// TIA Portal project "Game" (V18)

(* hardware
DEVICE "S7-1200 station_1"  S7-1200 Station
   slot 0: "Rack_0"  S7-1200 Rack  Rack  V1.0
   slot 1: "PLC_1"  CPU 1215C DC/DC/DC  6ES7 215-1AG40-0XB0  V4.4
DEVICE "PC-System_1"  SIMATIC PC station
   slot 0: "SIMATIC PC station"  Rail  SIMATIC PC-Station  V1.0
      slot 125: "Stationmanager"  Station_Manager  V6.0.4
   slot 1: "IE general_1"  IE General  IE_CP  V8.2.0
   slot 2: "HMI_RT_1"  WinCC RT Advanced  6AV2 104-0xxxx-xxxx  16.0.0.0
      slot 33792: "Computer interface"  Host interface
*)

// ===== PLC "PLC_1"  CPU 1215C DC/DC/DC =====

VAR_GLOBAL   // PLC tag table "Default tag table"
   "System_Byte" AT %MB1 : Byte;   // System Byte used for diagnostics or system status.
   "FirstScan" AT %M1.0 : Bool;   // Indicates the first scan of the PLC program.
   "DiagStatusUpdate" AT %M1.1 : Bool;   // Trigger for updating diagnostic status.
   "AlwaysTRUE" AT %M1.2 : Bool;   // Always holds the value TRUE.
   "AlwaysFALSE" AT %M1.3 : Bool;   // Always holds the value FALSE.
   "Clock_Byte" AT %MB0 : Byte;   // System clock byte for generating clock pulses.
   "Clock_10Hz" AT %M0.0 : Bool;   // 10 Hz clock pulse for timing operations.
   "Clock_5Hz" AT %M0.1 : Bool;   // 5 Hz clock pulse for timing operations.
   "Clock_2.5Hz" AT %M0.2 : Bool;   // 2.5 Hz clock pulse for timing operations.
   "Clock_2Hz" AT %M0.3 : Bool;   // 2 Hz clock pulse for timing operations.
   "Clock_1.25Hz" AT %M0.4 : Bool;   // 1.25 Hz clock pulse for timing operations.
   "Clock_1Hz" AT %M0.5 : Bool;   // 1 Hz clock pulse for timing operations.
   "Clock_0.625Hz" AT %M0.6 : Bool;   // 0.625 Hz clock pulse for timing operations.
   "Clock_0.5Hz" AT %M0.7 : Bool;   // 0.5 Hz clock pulse for timing operations.
   "lifebit" AT %M5.0 : Bool;   // Life bit toggled for system health monitoring.
   "Tag_1" AT %MW11 : Int;   // Temporary tag for integer calculations.
   "Tag_2" AT %MW12 : Word;   // Temporary tag for word calculations.
   "Tag_3" AT %M14.0 : Bool;   // Auxiliary flag for custom logic.
   "Tag_4" AT %MW4 : Word;   // Temporary tag for word operations.
   "draw number" AT %M20.0 : Bool;   // Trigger for generating random numbers.
   "Tag_6" AT %M100.0 : Bool;   // Auxiliary flag for random number validation.
   "temp int" AT %MW1 : Int;   // Temporary integer for calculations.
   "new game" AT %M15.0 : Bool;   // Signal to initialize a new game.
   "Tag_5" AT %M100.1 : Bool;   // Auxiliary flag for game initialization.
   "Tag_7" AT %M61.0 : Bool;   // Auxiliary signal for internal processing.
   "Tag_8" AT %M16.0 : Bool;   // Auxiliary signal for click detection.
   "Tag_9" AT %M16.1 : Bool;   // Auxiliary signal for click detection.
   "Tag_10" AT %M120.1 : Bool;   // Auxiliary signal for internal processing.
   "Tag_11" AT %M45.0 : Bool;   // Flag for triggering game logic.
   "Tag_12" AT %M45.1 : Bool;   // Auxiliary signal for additional logic.
   "reset limit" AT %M50.0 : Bool;   // Resets the field discovery limit.
   "start timer" AT %M40.0 : Bool;   // Starts the timer for incorrect moves.
   "start timer 2" AT %M40.1 : Bool;   // Starts the timer for correct moves.
   "running" AT %M10.5 : Bool;   // Indicates that the game is currently running.
   "win" AT %M10.6 : Bool;   // Signals that the game has been won.
   "Click1" AT %M65.0 : Bool;   // Signal for the first tile click.
   "Click2" AT %M65.1 : Bool;   // Signal for the second tile click.
   "Click3" AT %M65.2 : Bool;   // Signal for the third tile click.
   "Click4" AT %M65.3 : Bool;   // Signal for the fourth tile click.
   "Click5" AT %M65.4 : Bool;   // Signal for the fifth tile click.
   "Click6" AT %M65.5 : Bool;   // Signal for the sixth tile click.
   "Click7" AT %M65.6 : Bool;   // Signal for the seventh tile click.
   "Click8" AT %M65.7 : Bool;   // Signal for the eighth tile click.
   "Click9" AT %M66.0 : Bool;   // Signal for the ninth tile click.
   "Click10" AT %M66.1 : Bool;   // Signal for the tenth tile click.
   "Click11" AT %M66.2 : Bool;   // Signal for the eleventh tile click.
   "Click12" AT %M66.3 : Bool;   // Signal for the twelfth tile click.
   "Click13" AT %M66.4 : Bool;   // Signal for the thirteenth tile click.
   "Click14" AT %M66.5 : Bool;   // Signal for the fourteenth tile click.
   "Click15" AT %M66.6 : Bool;   // Signal for the fifteenth tile click.
   "Click16" AT %M66.7 : Bool;   // Signal for the sixteenth tile click.
END_VAR

DATA_BLOCK "Data_block_1"   // DB1
{ S7_Optimized_Access := 'TRUE' }
VERSION : 0.1
   VAR
      "time" : DTL;   // Current date and time used for generating random numbers.
      time2 : Time_Of_Day;   // Converted time of day extracted from the current system time.
      "time on udint" : UDInt;   // System time in unsigned double integer format for easier calculations.
      "tile array hidden" : Array[1..16] of Int;   // Stores the hidden values for each tile in the game.
      "tile array" : Array[1..16] of Int;   // Stores the currently revealed values for each tile.
      "guess tiles" : Array[1..16] of Int;   // Used to track player's guesses during the game
      "random number" : Int;   // Holds the latest randomly generated number for assigning tiles.
      "random numbers" : Array[1..16] of Int;   // Array of all unique randomly generated numbers for the game tiles.
      "array filled" : Bool;   // Indicates whether the tile array hidden is fully initialized.
      "number of moves" : Int;   // Tracks the total number of moves made by the player.
      "click detection" : Array[1..16] of Bool;   // Detects if a tile has been clicked by the player.
      "click detection2" : Array[1..16] of Bool;   // Additional array for detecting tile clicks used during validation.
      "field discovery limit" : Int;   // Counts the number of fields discovered by the player during a turn.
      "end of incorrect move" : Bool;   // Signals the end of an incorrect move.
      "end of correct move" : Bool;   // Signals the end of a correct move.
      "comparison mode" : Bool;   // Enables or disables the comparison logic between selected tiles.
      value1 : Int;   // The value of the first selected tile during a player's turn.
      value2 : Int;   // The value of the second selected tile during a player's turn.
      "value1 idx" : Int;   // The index of the first selected tile in the tile array.
      "value2 idx" : Int;   // The index of the second selected tile in the tile array.
      flag1 : Bool;   // Trigger used for checking game logic events like tile selection.
      flag2 : Bool;   // Additional trigger for handling specific game logic.
   END_VAR
BEGIN
END_DATA_BLOCK

// folder: System blocks/Program resources

DATA_BLOCK "IEC_Counter_0_DB"   // DB2
{ S7_Optimized_Access := 'TRUE' }
AUTHOR : Simatic
FAMILY : IEC
NAME : CNTR
VERSION : 1.0
// stored: InstanceOfName IEC_COUNTER
"IEC_COUNTER"
BEGIN
END_DATA_BLOCK

DATA_BLOCK "IEC_Timer_0_DB_2"   // DB4
{ S7_Optimized_Access := 'TRUE' }
AUTHOR : Simatic
FAMILY : IEC
NAME : IEC_TMR
VERSION : 1.0
// stored: InstanceOfName IEC_TIMER
"IEC_TIMER"
BEGIN
END_DATA_BLOCK

DATA_BLOCK "IEC_Timer_0_DB"   // DB5
{ S7_Optimized_Access := 'TRUE' }
AUTHOR : Simatic
FAMILY : IEC
NAME : IEC_TMR
VERSION : 1.0
// stored: InstanceOfName IEC_TIMER
"IEC_TIMER"
BEGIN
END_DATA_BLOCK

// folder: (top level)

FUNCTION "board filling SCL" : Void   // FC6, SCL
TITLE = board filling SCL
{ S7_Optimized_Access := 'TRUE' }
AUTHOR : krist
VERSION : 0.1
// Generating and placing random numbers on the game board.
   VAR_TEMP
      new : Bool;
      temp1 : Int;
      temp2 : Int;
      temp3 : Int;
      temp4 : Int;
   END_VAR
BEGIN
   #temp2 := 1;  // Iniciē mainīgo, kas skaita aizpildītās vērtības "random numbers" masīvā

   // Galvenais cikls, kas atkārto procesu 8 reizes
   FOR #temp1 := 1 TO 8 DO

       // Pārbauda, vai izlozētais skaitlis jau ir izmantots
       #"new" := FALSE;
       WHILE #"new" <> TRUE DO

           // Izveido nejaušu skaitli, izmantojot sistēmas laiku
           "Tag_1" := RD_LOC_T("Data_block_1"."time");
           "Data_block_1".time2 := DTL_TO_TOD("Data_block_1"."time");
           "Data_block_1"."time on udint" := TOD_TO_UDINT("Data_block_1".time2);
           "Data_block_1"."random number" := "Data_block_1"."time on udint" MOD 16;  // Ģenerē nejaušu skaitli starp 0 un 15
           "Data_block_1"."random number" += 1;  // Pielāgo, lai intervāls būtu no 1 līdz 16

           #"new" := TRUE;  // Pieņem, ka skaitlis ir jauns

           // Pārbauda, vai skaitlis jau eksistē "random numbers" masīvā
           FOR #temp3 := 1 TO 16 DO
               IF "Data_block_1"."random number" = "Data_block_1"."random numbers"[#temp3] THEN
                   #"new" := FALSE;  // Ja skaitlis eksistē, atkārto ģenerēšanas procesu
                   EXIT;
               END_IF;
           END_FOR;

       END_WHILE;

       // Piešķir nejaušo vērtību "tile array hidden" un saglabā "random numbers" masīvā
       "Data_block_1"."tile array hidden"["Data_block_1"."random number"] := #temp1;
       "Data_block_1"."random numbers"[#temp2] := "Data_block_1"."random number";
       #temp2 += 1;  // Palielina aizpildīto vērtību skaitītāju

       // Pārbauda, vai visi 16 skaitļi ir aizpildīti
       IF #temp2 = 16 THEN
           FOR #temp4 := 1 TO 16 DO
               IF "Data_block_1"."tile array hidden"[#temp4] = 0 THEN
                   "Data_block_1"."tile array hidden"[#temp4] := #temp1;  // Aizpilda atlikušo vietu masīvā
                   EXIT;
               END_IF;
           END_FOR;
           EXIT;  // Iziet no galvenā cikla, ja visi skaitļi ir aizpildīti
       END_IF;

       // Pārbauda, vai izlozētais skaitlis jau ir izmantots (otra izloze)
       #"new" := FALSE;
       WHILE #"new" <> TRUE DO

           // Izveido nejaušu skaitli, izmantojot sistēmas laiku
           "Tag_1" := RD_LOC_T("Data_block_1"."time");
           "Data_block_1".time2 := DTL_TO_TOD("Data_block_1"."time");
           "Data_block_1"."time on udint" := TOD_TO_UDINT("Data_block_1".time2);
           "Data_block_1"."random number" := "Data_block_1"."time on udint" MOD 15;  // Ģenerē nejaušu skaitli starp 0 un 14
           "Data_block_1"."random number" += 1;  // Pielāgo, lai intervāls būtu no 1 līdz 15

           #"new" := TRUE;  // Pieņem, ka skaitlis ir jauns

           // Pārbauda, vai skaitlis jau eksistē "random numbers" masīvā
           FOR #temp3 := 1 TO 16 DO
               IF "Data_block_1"."random number" = "Data_block_1"."random numbers"[#temp3] THEN
                   #"new" := FALSE;  // Ja skaitlis eksistē, atkārto ģenerēšanas procesu
                   EXIT;
               END_IF;
           END_FOR;

       END_WHILE;

       // Piešķir nejaušo vērtību "tile array hidden" un saglabā "random numbers" masīvā
       "Data_block_1"."tile array hidden"["Data_block_1"."random number"] := #temp1;
       "Data_block_1"."random numbers"[#temp2] := "Data_block_1"."random number";
       #temp2 += 1;  // Palielina aizpildīto vērtību skaitītāju

   END_FOR;

   // Atzīmē, ka masīvs ir pilnībā aizpildīts
   "Data_block_1"."array filled" := true;
END_FUNCTION

FUNCTION "clearing memory SCL" : Void   // FC7, SCL
TITLE = clearing memory SCL
{ S7_Optimized_Access := 'TRUE' }
AUTHOR : krist
VERSION : 0.1
// Clearing the game arrays and restoring the initial state
   VAR_TEMP
      temp : Int;
   END_VAR
BEGIN
   // Inicializē masīvus un mainīgos
   FOR #temp := 1 TO 16 DO
       "Data_block_1"."tile array"[#temp] := 0;           // Notīra "tile array" masīvu, uzstādot vērtības uz 0
       "Data_block_1"."tile array hidden"[#temp] := 0;    // Notīra "tile array hidden" masīvu, uzstādot vērtības uz 0
       "Data_block_1"."random numbers"[#temp] := 0;       // Notīra "random numbers" masīvu, uzstādot vērtības uz 0
       "Data_block_1"."click detection"[#temp] := 0;      // Notīra "click detection" masīvu, uzstādot vērtības uz 0
   END_FOR;

   // Inicializē citus parametrus
   "Data_block_1"."array filled" := FALSE;   // Norāda, ka masīvs nav aizpildīts
   "Data_block_1"."number of moves" := 0;    // Uzstāda gājienu skaitu uz 0
   "Data_block_1".value1 := 0;               // Notīra vērtību 1
   "Data_block_1".value2 := 0;               // Notīra vērtību 2
   "Data_block_1"."value1 idx" := 0;         // Notīra pirmā elementa indeksu
   "Data_block_1"."value2 idx" := 0;         // Notīra otrā elementa indeksu

   "Data_block_1"."comparison mode" := FALSE; // Izslēdz salīdzināšanas režīmu
   "win" := FALSE;                            // Norāda, ka spēle vēl nav uzvarēta
END_FUNCTION

FUNCTION "game SCL" : Void   // FC8, SCL
TITLE = game SCL
{ S7_Optimized_Access := 'TRUE' }
AUTHOR : krist
VERSION : 0.1
// The core logic of the game, including click processing and comparison.
   VAR_TEMP
      first : Int;
      second : Int;
   END_VAR
BEGIN

   "reset limit" := FALSE;  // Atjaunot limitu tiek atslēgts

   // Pārbaude, vai "field discovery limit" ir mazāks vai vienāds ar 2 un "Tag_11" ir TRUE
   IF "Data_block_1"."field discovery limit" <= 2 AND "Tag_11" THEN
       // Pārbauda katru elementu "click detection2" masīvā
       FOR #first := 1 TO 16 DO
           IF "Data_block_1"."click detection2"[#first] = TRUE AND "Data_block_1".value1 = 0 THEN
               EXIT;  // Iziet no cikla, ja atklāts klikšķis un vērtība 1 ir 0
           END_IF;
       END_FOR;

       // Apstrādā klikšķus un saglabā vērtības
       FOR #first := 1 TO 16 DO
           IF "Data_block_1"."click detection2"[#first] = TRUE THEN
               "Data_block_1"."tile array"[#first] := "Data_block_1"."tile array hidden"[#first];  // Atklāj slēpto elementu

               IF "Data_block_1".value1 = 0 THEN
                   "Data_block_1".value1 := "Data_block_1"."tile array"[#first];  // Saglabā pirmo vērtību
                   "Data_block_1"."value1 idx" := #first;  // Saglabā pirmā elementa indeksu
               END_IF;

               "Data_block_1".value2 := "Data_block_1"."tile array"[#first];  // Saglabā otro vērtību
               "Data_block_1"."value2 idx" := #first;  // Saglabā otrā elementa indeksu
           END_IF;
       END_FOR;
   END_IF;

   // Aktivizē trigeri, ja "field discovery limit" ir vienāds ar 2
   "R_TRIG_DB"(CLK := "Data_block_1"."field discovery limit" = 2,
               Q => "Data_block_1".flag1);

   // Ja trigeris aktivizēts, palielina gājienu skaitu
   IF "Data_block_1".flag1 = TRUE THEN
       "Data_block_1"."number of moves" += 1;

       // Pārbauda, vai vērtības ir vienādas
       IF "Data_block_1".value1 = "Data_block_1".value2 THEN
           "start timer 2" := TRUE;  // Aktivizē otro taimeri
       ELSE
           "start timer" := TRUE;  // Aktivizē pirmo taimeri
       END_IF;
   END_IF;

   // Apstrādā nepareizo gājienu
   IF "Data_block_1"."end of incorrect move" THEN
       "start timer" := FALSE;  // Izslēdz taimeri

       // Atiestata klikšķu izvēlētās vērtības un pozīcijas
       "Data_block_1"."tile array"["Data_block_1"."value1 idx"] := 0;
       "Data_block_1"."tile array"["Data_block_1"."value2 idx"] := 0;
       "Data_block_1".value1 := 0;
       "Data_block_1".value2 := 0;
       "Data_block_1"."value1 idx" := 0;
       "Data_block_1"."value2 idx" := 0;

       "reset limit" := TRUE;  // Aktivizē limitu
   END_IF;

   // Apstrādā pareizo gājienu
   IF "Data_block_1"."end of correct move" THEN
       "start timer 2" := FALSE;  // Izslēdz otro taimeri

       // Atiestata klikšķu izvēlētās vērtības un pozīcijas
       "Data_block_1".value1 := 0;
       "Data_block_1".value2 := 0;
       "Data_block_1"."value1 idx" := 0;
       "Data_block_1"."value2 idx" := 0;

       "reset limit" := TRUE;  // Aktivizē limitu
   END_IF;

   // Pārbauda, vai visi elementi ir atklāti
   FOR #second := 1 TO 16 DO
       IF "Data_block_1"."tile array"[#second] = 0 THEN
           EXIT;  // Iziet, ja kāds elements nav atklāts
       END_IF;

       IF #second = 16 THEN
           "win" := TRUE;  // Uzvaras nosacījums
       END_IF;
   END_FOR;

   // Atiestata klikšķu detekcijas statusu
   FOR #first := 1 TO 16 DO
       "Data_block_1"."click detection2"[#first] := FALSE;
   END_FOR;
END_FUNCTION

FUNCTION "button operation LAD" : Void   // FC9, LAD
TITLE = button operation LAD
{ S7_Optimized_Access := 'TRUE' }
AUTHOR : krist
VERSION : 0.1
// Detecting clicks and passing them to game logic.
   VAR_TEMP   // added for the SCL form of the ladder/FBD networks
      _w1 : Bool;
      _w2 : Bool;
      _w3 : Bool;
      _w4 : Bool;
      _w5 : Bool;
      _w6 : Bool;
      _w7 : Bool;
      _w8 : Bool;
      _w9 : Bool;
      _w10 : Bool;
      _w11 : Bool;
      _w12 : Bool;
      _w13 : Bool;
      _w14 : Bool;
      _w15 : Bool;
      _w16 : Bool;
      _w17 : Bool;
      _w18 : Bool;
   END_VAR
BEGIN

REGION Network 1: Additional array for detecting tile clicks used during validation.
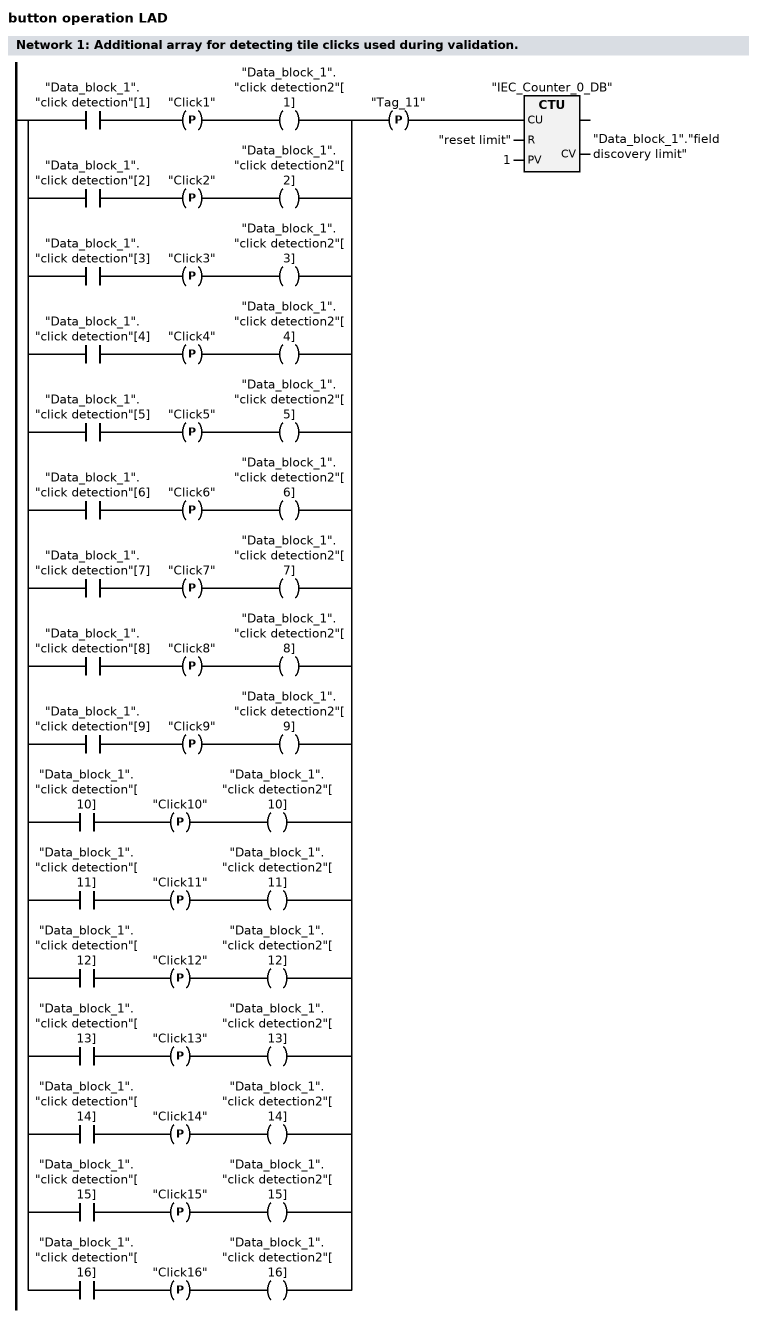
   #_w1 := "Data_block_1"."click detection"[1] AND NOT "Click1";   // rising edge
   "Click1" := "Data_block_1"."click detection"[1];
   "Data_block_1"."click detection2"[1] := #_w1;
   #_w2 := "Data_block_1"."click detection"[2] AND NOT "Click2";   // rising edge
   "Click2" := "Data_block_1"."click detection"[2];
   "Data_block_1"."click detection2"[2] := #_w2;
   #_w3 := "Data_block_1"."click detection"[3] AND NOT "Click3";   // rising edge
   "Click3" := "Data_block_1"."click detection"[3];
   "Data_block_1"."click detection2"[3] := #_w3;
   #_w4 := "Data_block_1"."click detection"[4] AND NOT "Click4";   // rising edge
   "Click4" := "Data_block_1"."click detection"[4];
   "Data_block_1"."click detection2"[4] := #_w4;
   #_w5 := "Data_block_1"."click detection"[5] AND NOT "Click5";   // rising edge
   "Click5" := "Data_block_1"."click detection"[5];
   "Data_block_1"."click detection2"[5] := #_w5;
   #_w6 := "Data_block_1"."click detection"[6] AND NOT "Click6";   // rising edge
   "Click6" := "Data_block_1"."click detection"[6];
   "Data_block_1"."click detection2"[6] := #_w6;
   #_w7 := "Data_block_1"."click detection"[7] AND NOT "Click7";   // rising edge
   "Click7" := "Data_block_1"."click detection"[7];
   "Data_block_1"."click detection2"[7] := #_w7;
   #_w8 := "Data_block_1"."click detection"[8] AND NOT "Click8";   // rising edge
   "Click8" := "Data_block_1"."click detection"[8];
   "Data_block_1"."click detection2"[8] := #_w8;
   #_w9 := "Data_block_1"."click detection"[9] AND NOT "Click9";   // rising edge
   "Click9" := "Data_block_1"."click detection"[9];
   "Data_block_1"."click detection2"[9] := #_w9;
   #_w10 := "Data_block_1"."click detection"[10] AND NOT "Click10";   // rising edge
   "Click10" := "Data_block_1"."click detection"[10];
   "Data_block_1"."click detection2"[10] := #_w10;
   #_w11 := "Data_block_1"."click detection"[11] AND NOT "Click11";   // rising edge
   "Click11" := "Data_block_1"."click detection"[11];
   "Data_block_1"."click detection2"[11] := #_w11;
   #_w12 := "Data_block_1"."click detection"[12] AND NOT "Click12";   // rising edge
   "Click12" := "Data_block_1"."click detection"[12];
   "Data_block_1"."click detection2"[12] := #_w12;
   #_w13 := "Data_block_1"."click detection"[13] AND NOT "Click13";   // rising edge
   "Click13" := "Data_block_1"."click detection"[13];
   "Data_block_1"."click detection2"[13] := #_w13;
   #_w14 := "Data_block_1"."click detection"[14] AND NOT "Click14";   // rising edge
   "Click14" := "Data_block_1"."click detection"[14];
   "Data_block_1"."click detection2"[14] := #_w14;
   #_w15 := "Data_block_1"."click detection"[15] AND NOT "Click15";   // rising edge
   "Click15" := "Data_block_1"."click detection"[15];
   "Data_block_1"."click detection2"[15] := #_w15;
   #_w16 := "Data_block_1"."click detection"[16] AND NOT "Click16";   // rising edge
   "Click16" := "Data_block_1"."click detection"[16];
   "Data_block_1"."click detection2"[16] := #_w16;
   #_w17 := #_w1 OR #_w2 OR #_w3 OR #_w4 OR #_w5 OR #_w6 OR #_w7 OR #_w8 OR #_w9 OR #_w10 OR #_w11 OR #_w12 OR #_w13 OR #_w14 OR #_w15 OR #_w16;
   #_w18 := #_w17 AND NOT "Tag_11";   // rising edge
   "Tag_11" := #_w17;
   "IEC_Counter_0_DB".CTU(CU := #_w18,
                          R := "reset limit",
                          PV := 1,
                          CV => "Data_block_1"."field discovery limit");
END_REGION
END_FUNCTION

FUNCTION "timer LAD" : Void   // FC10, LAD
TITLE = timer LAD
{ S7_Optimized_Access := 'TRUE' }
VERSION : 0.1
// Timer functions for handling correct and incorrect moves.
BEGIN

REGION Network 1: Signals the end of an incorrect move.
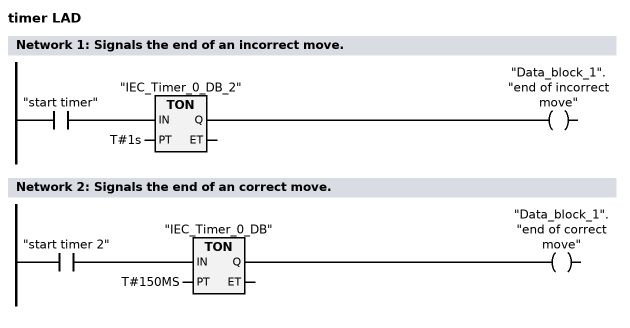
   "IEC_Timer_0_DB_2".TON(IN := "start timer", PT := T#1s);
   "Data_block_1"."end of incorrect move" := "IEC_Timer_0_DB_2".Q;
END_REGION

REGION Network 2: Signals the end of an correct move.
   "IEC_Timer_0_DB".TON(IN := "start timer 2", PT := T#150MS);
   "Data_block_1"."end of correct move" := "IEC_Timer_0_DB".Q;
END_REGION
END_FUNCTION

ORGANIZATION_BLOCK "Main"   // OB1, LAD, ProgramCycle
TITLE = "Main Program Sweep (Cycle)"
{ S7_Optimized_Access := 'TRUE' }
VERSION : 0.1
   VAR_INPUT
      Initial_Call : Bool;   // Initial call of this OB
      Remanence : Bool;   // =True, if remanent data are available
   END_VAR
   VAR_TEMP   // added for the SCL form of the ladder/FBD networks
      _w1 : Bool;
      _w2 : Bool;
   END_VAR
BEGIN

REGION Network 1
   // indicates systems activity
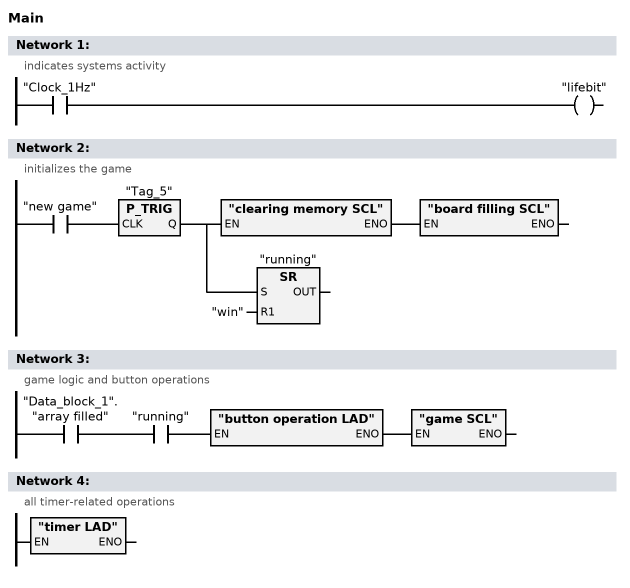
   RUNG wire#powerrail
      Contact( "Clock_1Hz" )
      Coil( "lifebit" )
   END_RUNG
   // the same network as SCL:
   "lifebit" := "Clock_1Hz";
END_REGION

REGION Network 2
   // initializes the game
   RUNG wire#powerrail
      Contact( "new game" )
      P_Trig( "Tag_5" )
      wire#w1
      "clearing memory SCL"()
      "board filling SCL"()
   END_RUNG
   RUNG wire#w1
      S_SR(operand := "running", r1 := "win")
   END_RUNG
   // the same network as SCL:
   #_w1 := "new game" AND NOT "Tag_5";   // rising edge
   "Tag_5" := "new game";
   "clearing memory SCL"(EN := #_w1, ENO => #_w2);
   IF #_w2 THEN "board filling SCL"(); END_IF;
   IF #_w1 THEN
       "running" := TRUE;   // SR flip-flop
   END_IF;
   IF "win" THEN "running" := FALSE; END_IF;
END_REGION

REGION Network 3
   // game logic and button operations
   RUNG wire#powerrail
      Contact( "Data_block_1"."array filled" )
      Contact( "running" )
      "button operation LAD"()
      "game SCL"()
   END_RUNG
   // the same network as SCL:
   "button operation LAD"(EN := "Data_block_1"."array filled" AND "running", ENO => #_w1);
   IF #_w1 THEN "game SCL"(); END_IF;
END_REGION

REGION Network 4
   // all timer-related operations
   RUNG wire#powerrail
      "timer LAD"()
   END_RUNG
   // the same network as SCL:
   "timer LAD"();
END_REGION
END_ORGANIZATION_BLOCK

(* ===== HMI "HMI_RT_1" =====
system functions are stored by id; their names below are inferred from use
connection "HMI_Connection_1": ETHERNET, S7_1200_OMS

HMI tags "Default tag table"
   "lifebit" : Bool = PLC lifebit AT %M5.0, 100 ms
   "wylosuj liczbe" : Bool = PLC "draw number" AT %M20.0, 100 ms
   "Data_block_1_wylosowana liczba" : Int = PLC Data_block_1."random number", 100 ms
   "Data_block_1_tile array{1}" : Int = PLC Data_block_1."tile array"[1], 100 ms
   "Data_block_1_tile array{2}" : Int = PLC Data_block_1."tile array"[2], 100 ms
   "Data_block_1_tile array{3}" : Int = PLC Data_block_1."tile array"[3], 100 ms
   "Data_block_1_tile array{4}" : Int = PLC Data_block_1."tile array"[4], 100 ms
   "Data_block_1_tile array{5}" : Int = PLC Data_block_1."tile array"[5], 100 ms
   "Data_block_1_tile array{6}" : Int = PLC Data_block_1."tile array"[6], 100 ms
   "Data_block_1_tile array{7}" : Int = PLC Data_block_1."tile array"[7], 100 ms
   "Data_block_1_tile array{8}" : Int = PLC Data_block_1."tile array"[8], 100 ms
   "Data_block_1_tile array{9}" : Int = PLC Data_block_1."tile array"[9], 100 ms
   "Data_block_1_tile array{10}" : Int = PLC Data_block_1."tile array"[10], 100 ms
   "Data_block_1_tile array{11}" : Int = PLC Data_block_1."tile array"[11], 100 ms
   "Data_block_1_tile array{12}" : Int = PLC Data_block_1."tile array"[12], 100 ms
   "Data_block_1_tile array{13}" : Int = PLC Data_block_1."tile array"[13], 100 ms
   "Data_block_1_tile array{14}" : Int = PLC Data_block_1."tile array"[14], 100 ms
   "Data_block_1_tile array{15}" : Int = PLC Data_block_1."tile array"[15], 100 ms
   "Data_block_1_tile array{16}" : Int = PLC Data_block_1."tile array"[16], 100 ms
   "Nowa gra" : Bool = PLC "new game" AT %M15.0, 100 ms
   "Data_block_1_detect click{1}" : Bool = PLC Data_block_1."click detection"[1], 1 s
   "Data_block_1_detect click{2}" : Bool = PLC Data_block_1."click detection"[2], 1 s
   "Data_block_1_detect click{3}" : Bool = PLC Data_block_1."click detection"[3], 1 s
   "Data_block_1_detect click{4}" : Bool = PLC Data_block_1."click detection"[4], 1 s
   "Data_block_1_detekcja klikniec{5}" : Bool = PLC Data_block_1."click detection"[5], 1 s
   "Data_block_1_detekcja klikniec{6}" : Bool = PLC Data_block_1."click detection"[6], 1 s
   "Data_block_1_detekcja klikniec{7}" : Bool = PLC Data_block_1."click detection"[7], 1 s
   "Data_block_1_detekcja klikniec{8}" : Bool = PLC Data_block_1."click detection"[8], 1 s
   "Data_block_1_detekcja klikniec{9}" : Bool = PLC Data_block_1."click detection"[9], 1 s
   "Data_block_1_detect click{10}" : Bool = PLC Data_block_1."click detection"[10], 1 s
   "Data_block_1_detect click{11}" : Bool = PLC Data_block_1."click detection"[11], 1 s
   "Data_block_1_detect click{12}" : Bool = PLC Data_block_1."click detection"[12], 1 s
   "Data_block_1_detect click{13}" : Bool = PLC Data_block_1."click detection"[13], 1 s
   "Data_block_1_detect click{14}" : Bool = PLC Data_block_1."click detection"[14], 1 s
   "Data_block_1_detect click{15}" : Bool = PLC Data_block_1."click detection"[15], 1 s
   "Data_block_1_detect click{16}" : Bool = PLC Data_block_1."click detection"[16], 1 s
   "Data_block_1_ilosc ruchow" : Int = PLC Data_block_1."number of moves", 1 s
   "reset limitu" : Bool = PLC "reset limit" AT %M50.0, 1 s
   "win" : Bool = PLC win AT %M10.6, 1 s

screen "Game" 1024x768
   Circle "Circle_1" at 394,112 size 48x48
      Appearance <- "lifebit"
   Button "Button_2" at 571,63 size 96x32; TextOff 'New Game'
      on Press: function_b14e0dd5("Nowa gra", 0); function_b14e0dd5("reset limitu", 0)
   Group "Group" at 309,182 size 100x100; FormatPattern 9999999
   Group "Group_1" at 409,182 size 100x100; FormatPattern 9999999
   Group "Group_2" at 509,182 size 100x100; FormatPattern 9999999
   Group "Group_3" at 609,182 size 100x100; FormatPattern 9999999
   Group "Group_4" at 309,282 size 100x100; FormatPattern 9999999
   Group "Group_5" at 409,282 size 100x100; FormatPattern 9999999
   Group "Group_6" at 509,282 size 100x100; FormatPattern 9999999
   Group "Group_7" at 609,282 size 100x100; FormatPattern 9999999
   Group "Group_8" at 309,382 size 100x100; FormatPattern 9999999
   Group "Group_9" at 409,382 size 100x100; FormatPattern 9999999
   Group "Group_10" at 509,382 size 100x100; FormatPattern 9999999
   Group "Group_11" at 609,382 size 100x100; FormatPattern 9999999
   Group "Group_12" at 309,482 size 100x100; FormatPattern 9999999
   Group "Group_13" at 409,482 size 100x100; FormatPattern 9999999
   Group "Group_14" at 509,482 size 100x100; FormatPattern 9999999
   Group "Group_15" at 609,482 size 100x100; FormatPattern 9999999
   IOField "I/O field_1" at 453,63 size 96x32; FormatPattern 99999
      ProcessValue <- "Data_block_1_ilosc ruchow"
   TextField "Text field_1" at 388,63 size 53x22; Text 'Moves'
   Group "Group_16" at 453,112 size 96x48
   IOField "I/O field_2" at 309,182 size 100x100; FormatPattern 99
      ProcessValue <- "Data_block_1_tile array{1}"
   Button "Button_1" at 309,182 size 100x100; TextOff '1'
      on Press: function_b14e0dd5("Data_block_1_detect click{1}", 0)
   IOField "I/O field_3" at 409,182 size 100x100; FormatPattern 99
      ProcessValue <- "Data_block_1_tile array{2}"
   Button "Button_3" at 409,182 size 100x100; TextOff 'Text'
      on Press: function_b14e0dd5("Data_block_1_detect click{2}", 0)
   IOField "I/O field_4" at 509,182 size 100x100; FormatPattern 99
      ProcessValue <- "Data_block_1_tile array{3}"
   Button "Button_4" at 509,182 size 100x100; TextOff 'Text'
      on Press: function_b14e0dd5("Data_block_1_detect click{3}", 0)
   IOField "I/O field_5" at 609,182 size 100x100; FormatPattern 99
      ProcessValue <- "Data_block_1_tile array{4}"
   Button "Button_5" at 609,182 size 100x100; TextOff 'Text'
      on Press: function_b14e0dd5("Data_block_1_detect click{4}", 0)
   IOField "I/O field_6" at 309,282 size 100x100; FormatPattern 99
      ProcessValue <- "Data_block_1_tile array{5}"
   Button "Button_6" at 309,282 size 100x100; TextOff 'Text'
      on Press: function_b14e0dd5("Data_block_1_detekcja klikniec{5}", 0)
   IOField "I/O field_7" at 409,282 size 100x100; FormatPattern 99
      ProcessValue <- "Data_block_1_tile array{6}"
   Button "Button_7" at 409,282 size 100x100; TextOff 'Text'
      on Press: function_b14e0dd5("Data_block_1_detekcja klikniec{6}", 0)
   IOField "I/O field_8" at 509,282 size 100x100; FormatPattern 99
      ProcessValue <- "Data_block_1_tile array{7}"
   Button "Button_8" at 509,282 size 100x100; TextOff 'Text'
      on Press: function_b14e0dd5("Data_block_1_detekcja klikniec{7}", 0)
   IOField "I/O field_9" at 609,282 size 100x100; FormatPattern 99
      ProcessValue <- "Data_block_1_tile array{8}"
   Button "Button_9" at 609,282 size 100x100; TextOff 'Text'
      on Press: function_b14e0dd5("Data_block_1_detekcja klikniec{8}", 0)
   IOField "I/O field_10" at 309,382 size 100x100; FormatPattern 99
      ProcessValue <- "Data_block_1_tile array{9}"
   Button "Button_10" at 309,382 size 100x100; TextOff 'Text'
      on Press: function_b14e0dd5("Data_block_1_detekcja klikniec{9}", 0)
   IOField "I/O field_11" at 409,382 size 100x100; FormatPattern 99
      ProcessValue <- "Data_block_1_tile array{10}"
   Button "Button_11" at 409,382 size 100x100; TextOff 'Text'
      on Press: function_b14e0dd5("Data_block_1_detect click{10}", 0)
   IOField "I/O field_12" at 509,382 size 100x100; FormatPattern 99
      ProcessValue <- "Data_block_1_tile array{11}"
   Button "Button_12" at 509,382 size 100x100; TextOff 'Text'
      on Press: function_b14e0dd5("Data_block_1_detect click{11}", 0)
   IOField "I/O field_13" at 609,382 size 100x100; FormatPattern 99
      ProcessValue <- "Data_block_1_tile array{12}"
   Button "Button_13" at 609,382 size 100x100; TextOff 'Text'
      on Press: function_b14e0dd5("Data_block_1_detect click{12}", 0)
   IOField "I/O field_14" at 309,482 size 100x100; FormatPattern 99
      ProcessValue <- "Data_block_1_tile array{13}"
   Button "Button_14" at 309,482 size 100x100; TextOff 'Text'
      on Press: function_b14e0dd5("Data_block_1_detect click{13}", 0)
   IOField "I/O field_15" at 409,482 size 100x100; FormatPattern 99
      ProcessValue <- "Data_block_1_tile array{14}"
   Button "Button_15" at 409,482 size 100x100; TextOff 'Text'
      on Press: function_b14e0dd5("Data_block_1_detect click{14}", 0)
   IOField "I/O field_16" at 509,482 size 100x100; FormatPattern 99
      ProcessValue <- "Data_block_1_tile array{15}"
   Button "Button_16" at 509,482 size 100x100; TextOff 'Text'
      on Press: function_b14e0dd5("Data_block_1_detect click{15}", 0)
   IOField "I/O field_17" at 609,482 size 100x100; FormatPattern 99
      ProcessValue <- "Data_block_1_tile array{16}"
   Button "Button_17" at 609,482 size 100x100; TextOff 'Text'
      on Press: function_b14e0dd5("Data_block_1_detect click{16}", 0)
   Rectangle "Rectangle_2" at 453,112 size 96x48
      Visibility <- "win"
   TextField "Text field_2" at 465,128 size 74x21; Text 'You Win'
      Visibility <- "win"
*)